PROGRAM ITInterruption
VAR
	//FB qui interrompent un tâche en cours de la structure via des signaux d'interruption - Alec 08.11.23
	balise : FB_Balise;			//gère la Balise et les visus qui lui sont associé 
	timeout: FB_Timeout;		//le temps du match arrive à sa fin
	restartTwincat : TC_Restart;//redémarre twincat
END_VAR

VAR_INPUT
	//interface - Alec 08.11.23
	IbStartBalise 		:BOOL; //Démarre le moteur de la balise
	IbMatchEnCours		:BOOL; //Match en cours
	IbStartVisuBalise	:BOOL; //Démarre la visu balise (à ne pas faire tourner pendant les matchs dans l'idéal car elle demande pas mal de ressource)
	IbRestartTwincat	:BOOL; //Redémarre twincat
	IbArretDetection	:BOOL; //Arrête la détection pendant que la variable est à TRUE
END_VAR

VAR_OUTPUT
	//Signaux d'interruption qui influencent le system - Alec 08.11.23
	QbStopMotion		:BOOL;	//Arrête les moteurs du robot 
	QbPauseMotion  		:BOOL;	//interrompt le déplacement du robot tant que la variable est à TRUE 
	QbResetMotion 		:BOOL;	//Fait un reset des moteurs en cas d'erreur 
	QbEndMatch 			:BOOL;	//Si _3_Match va en _8_EndMatch
	QbAbortTask			:BOOL;	//Arrête la tâche en cours (dépend de l'étape actuel de la structure)
								//si _1_INIT => recommence l'init
								//si _2_PREMATCH => retourne à l'init
								//si _6_INTERRUPTION => change la ligne actuelle du Tableau (changement de tâche)
END_VAR
VAR // added by the converter: edge detectors and wires of the graphical bodies
    _w1, _w2 : BOOL;
END_VAR

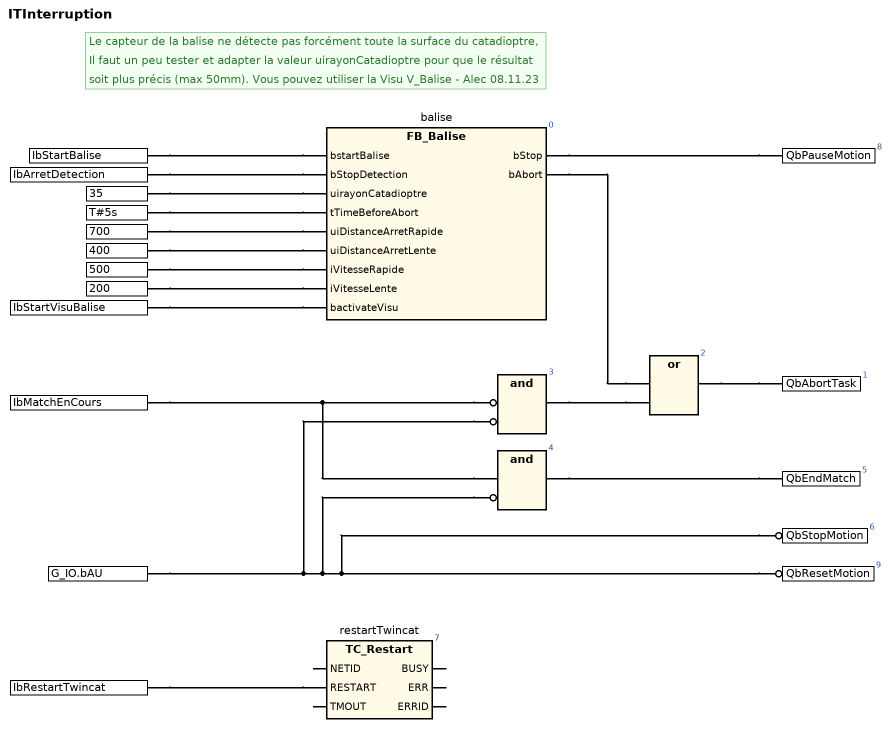
// Le capteur de la balise ne détecte pas forcément toute la surface du catadioptre,
// Il faut un peu tester et adapter la valeur uirayonCatadioptre pour que le résultat
// soit plus précis (max 50mm). Vous pouvez utiliser la Visu V_Balise - Alec 08.11.23
balise(
    bstartBalise := IbStartBalise,
    bStopDetection := IbArretDetection,
    uirayonCatadioptre := 35,
    tTimeBeforeAbort := T#5s,
    uiDistanceArretRapide := 700,
    uiDistanceArretLente := 400,
    iVitesseRapide := 500,
    iVitesseLente := 200,
    bactivateVisu := IbStartVisuBalise); // FB_Balise
QbAbortTask := _w1;
_w1 := balise.bAbort OR _w2;
_w2 := NOT IbMatchEnCours AND NOT G_IO.bAU;
QbEndMatch := IbMatchEnCours AND NOT G_IO.bAU;
QbStopMotion := NOT G_IO.bAU;
restartTwincat(RESTART := IbRestartTwincat); // TC_Restart
QbPauseMotion := balise.bStop;
QbResetMotion := NOT G_IO.bAU;

END_PROGRAM

(* stored: Version 1.1.0.1, ProductVersion 3.1.4024.12
   POU ITInterruption: Id {e85c749b-717a-437d-ba5d-2c10643297b7}, SpecialFunc None *)
